(* CoDeSys 2.3 export: SCODE_CODE.EXP *)

(* POU MNG_TCPIP/Helper functions/function blocks/SCODE_CODE, ST *)
FUNCTION SCODE_CODE : DWORD
(* Helper function: returns the lower word of error code *)
VAR_INPUT
	sc		: UDINT;
END_VAR
SCODE_CODE := 16#FFFF AND UDINT_TO_DWORD( sc );
END_FUNCTION
